REGION Network 93: 51.093 | n0093-ug7-el001-k30001_SN51 [3]
   RUNG wire#powerrail
      "FDBK_Error_n0093-ug7-el001-k30001_SN51_3"(Commissioning_bypass := "00_Commissioning"."n0093-ug7-el001-k30001_SN51", "FDBACK ERROR 1" := "FDBACK_=SG06+UG7.EL001-Q32801/Q32802".ERROR, "FDBACK ERROR 2" := "FDBACK_=SG06+UG7.EL001-Q32803/Q32804".ERROR, "FDBACK ERROR 3" := "FDBACK_=SG06+UG7.EL001-Q32901/Q32902".ERROR, "FDBACK ERROR 4" := "FDBACK_=SG06+UG7.EL001-Q32903/Q32904".ERROR, "FDBACK ERROR 5" :=, "FDBACK ERROR 6" :=, "FDBACK ERROR 7" :=, "FDBACK ERROR 8" :=, "Cumulative FDBACK" =>, "ERROR 1" => "03_FDBACK"."SG06+UG7.EL001-Q32802", "ERROR 2" => "03_FDBACK"."SG06+UG7.EL001-Q32804", "ERROR 3" => "03_FDBACK"."SG06+UG7.EL001-Q32902", "ERROR 4" => "03_FDBACK"."SG06+UG7.EL001-Q32904", "ERROR 5" =>, "ERROR 6" =>, "ERROR 7" =>, "ERROR 8" =>)
   END_RUNG
   // the same network as SCL:
   "FDBK_Error_n0093-ug7-el001-k30001_SN51_3"(Commissioning_bypass := "00_Commissioning"."n0093-ug7-el001-k30001_SN51",   // "03_FDBACK error"
                           "FDBACK ERROR 1" := "FDBACK_=SG06+UG7.EL001-Q32801/Q32802".ERROR,
                           "FDBACK ERROR 2" := "FDBACK_=SG06+UG7.EL001-Q32803/Q32804".ERROR,
                           "FDBACK ERROR 3" := "FDBACK_=SG06+UG7.EL001-Q32901/Q32902".ERROR,
                           "FDBACK ERROR 4" := "FDBACK_=SG06+UG7.EL001-Q32903/Q32904".ERROR,
                           "ERROR 1" => "03_FDBACK"."SG06+UG7.EL001-Q32802",
                           "ERROR 2" => "03_FDBACK"."SG06+UG7.EL001-Q32804",
                           "ERROR 3" => "03_FDBACK"."SG06+UG7.EL001-Q32902",
                           "ERROR 4" => "03_FDBACK"."SG06+UG7.EL001-Q32904");
END_REGION
END_FUNCTION

FUNCTION "07_Speed Control" : Void   // FC8, F_LAD
{ S7_Optimized_Access := 'TRUE' }
VERSION : 0.1
BEGIN

REGION Network 1: One network per sorter
END_REGION

REGION Network 2
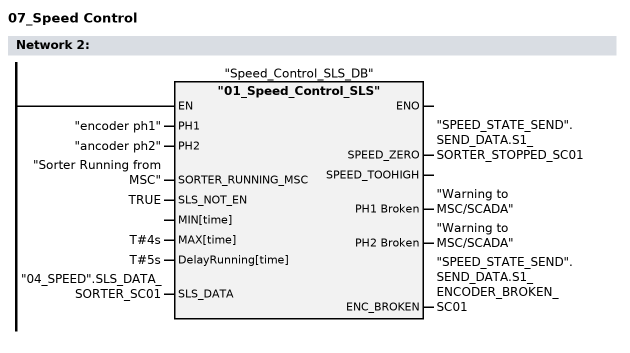
   RUNG wire#powerrail
      "Speed_Control_SLS_DB"(PH1 := "encoder ph1", PH2 := "ancoder ph2", SORTER_RUNNING_MSC := "Sorter Running from MSC", SLS_NOT_EN := TRUE, "MIN[time]" :=, "MAX[time]" := T#4s, "DelayRunning[time]" := T#5s, SLS_DATA := "04_SPEED".SLS_DATA_SORTER_SC01, SPEED_ZERO => "SPEED_STATE_SEND".SEND_DATA.S1_SORTER_STOPPED_SC01, SPEED_TOOHIGH =>, "PH1 Broken" => "Warning to MSC/SCADA", "PH2 Broken" => "Warning to MSC/SCADA", ENC_BROKEN => "SPEED_STATE_SEND".SEND_DATA.S1_ENCODER_BROKEN_SC01)
   END_RUNG
   // the same network as SCL:
   "Speed_Control_SLS_DB"(PH1 := "encoder ph1",   // "01_Speed_Control_SLS"
                          PH2 := "ancoder ph2",
                          SORTER_RUNNING_MSC := "Sorter Running from MSC",
                          SLS_NOT_EN := TRUE,
                          "MAX[time]" := T#4s,
                          "DelayRunning[time]" := T#5s,
                          SLS_DATA := "04_SPEED".SLS_DATA_SORTER_SC01,
                          SPEED_ZERO => "SPEED_STATE_SEND".SEND_DATA.S1_SORTER_STOPPED_SC01,
                          "PH1 Broken" => "Warning to MSC/SCADA",
                          "PH2 Broken" => "Warning to MSC/SCADA",
                          ENC_BROKEN => "SPEED_STATE_SEND".SEND_DATA.S1_ENCODER_BROKEN_SC01);
END_REGION
END_FUNCTION

FUNCTION "08_Gate Manager" : Void   // FC9, F_LAD
{ S7_Optimized_Access := 'TRUE' }
VERSION : 0.1
   VAR_TEMP
      temp_EXAMPLE_OPEN : Bool;
   END_VAR
BEGIN

REGION Network 1: Transfer Data from Speed Control
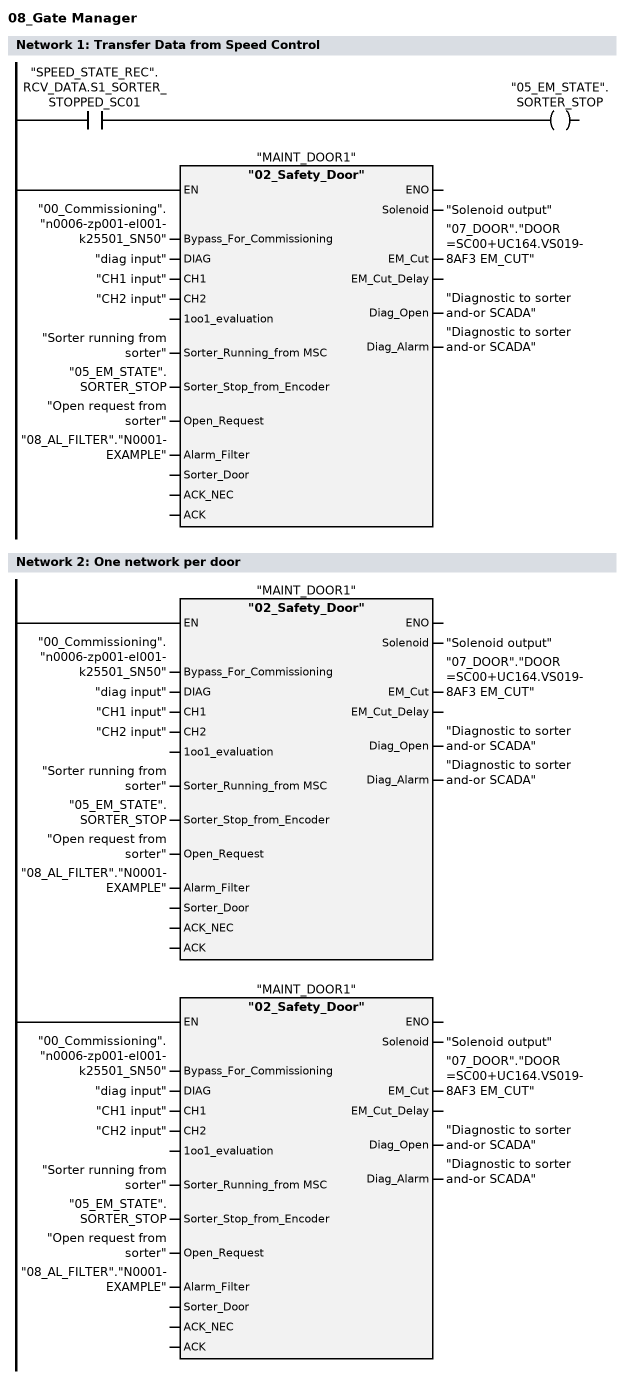
   RUNG wire#powerrail
      Contact( "SPEED_STATE_REC".RCV_DATA.S1_SORTER_STOPPED_SC01 )
      Coil( "05_EM_STATE".SORTER_STOP )
   END_RUNG
   RUNG wire#powerrail
      "MAINT_DOOR1"(Bypass_For_Commissioning := "00_Commissioning"."n0006-zp001-el001-k25501_SN50", DIAG := "diag input", CH1 := "CH1 input", CH2 := "CH2 input", "1oo1_evaluation" :=, "Sorter_Running_from MSC" := "Sorter running from sorter", Sorter_Stop_from_Encoder := "05_EM_STATE".SORTER_STOP, Open_Request := "Open request from sorter", Alarm_Filter := "08_AL_FILTER"."N0001-EXAMPLE", Sorter_Door :=, ACK_NEC :=, ACK :=, Solenoid => "Solenoid output", EM_Cut => "07_DOOR"."DOOR =SC00+UC164.VS019-8AF3 EM_CUT", EM_Cut_Delay =>, Diag_Open => "Diagnostic to sorter and-or SCADA", Diag_Alarm => "Diagnostic to sorter and-or SCADA")
   END_RUNG
   RUNG wire#powerrail
   END_RUNG
   // the same network as SCL:
   "05_EM_STATE".SORTER_STOP := "SPEED_STATE_REC".RCV_DATA.S1_SORTER_STOPPED_SC01;
   "MAINT_DOOR1"(Bypass_For_Commissioning := "00_Commissioning"."n0006-zp001-el001-k25501_SN50",   // "02_Safety_Door"
                 DIAG := "diag input",
                 CH1 := "CH1 input",
                 CH2 := "CH2 input",
                 "Sorter_Running_from MSC" := "Sorter running from sorter",
                 Sorter_Stop_from_Encoder := "05_EM_STATE".SORTER_STOP,
                 Open_Request := "Open request from sorter",
                 Alarm_Filter := "08_AL_FILTER"."N0001-EXAMPLE",
                 Solenoid => "Solenoid output",
                 EM_Cut => "07_DOOR"."DOOR =SC00+UC164.VS019-8AF3 EM_CUT",
                 Diag_Open => "Diagnostic to sorter and-or SCADA",
                 Diag_Alarm => "Diagnostic to sorter and-or SCADA");
END_REGION

REGION Network 2: One network per door
   RUNG wire#powerrail
      "MAINT_DOOR1"(Bypass_For_Commissioning := "00_Commissioning"."n0006-zp001-el001-k25501_SN50", DIAG := "diag input", CH1 := "CH1 input", CH2 := "CH2 input", "1oo1_evaluation" :=, "Sorter_Running_from MSC" := "Sorter running from sorter", Sorter_Stop_from_Encoder := "05_EM_STATE".SORTER_STOP, Open_Request := "Open request from sorter", Alarm_Filter := "08_AL_FILTER"."N0001-EXAMPLE", Sorter_Door :=, ACK_NEC :=, ACK :=, Solenoid => "Solenoid output", EM_Cut => "07_DOOR"."DOOR =SC00+UC164.VS019-8AF3 EM_CUT", EM_Cut_Delay =>, Diag_Open => "Diagnostic to sorter and-or SCADA", Diag_Alarm => "Diagnostic to sorter and-or SCADA")
   END_RUNG
   RUNG wire#powerrail
      "MAINT_DOOR1"(Bypass_For_Commissioning := "00_Commissioning"."n0006-zp001-el001-k25501_SN50", DIAG := "diag input", CH1 := "CH1 input", CH2 := "CH2 input", "1oo1_evaluation" :=, "Sorter_Running_from MSC" := "Sorter running from sorter", Sorter_Stop_from_Encoder := "05_EM_STATE".SORTER_STOP, Open_Request := "Open request from sorter", Alarm_Filter := "08_AL_FILTER"."N0001-EXAMPLE", Sorter_Door :=, ACK_NEC :=, ACK :=, Solenoid => "Solenoid output", EM_Cut => "07_DOOR"."DOOR =SC00+UC164.VS019-8AF3 EM_CUT", EM_Cut_Delay =>, Diag_Open => "Diagnostic to sorter and-or SCADA", Diag_Alarm => "Diagnostic to sorter and-or SCADA")
   END_RUNG
   // the same network as SCL:
   "MAINT_DOOR1"(Bypass_For_Commissioning := "00_Commissioning"."n0006-zp001-el001-k25501_SN50",   // "02_Safety_Door"
                 DIAG := "diag input",
                 CH1 := "CH1 input",
                 CH2 := "CH2 input",
                 "Sorter_Running_from MSC" := "Sorter running from sorter",
                 Sorter_Stop_from_Encoder := "05_EM_STATE".SORTER_STOP,
                 Open_Request := "Open request from sorter",
                 Alarm_Filter := "08_AL_FILTER"."N0001-EXAMPLE",
                 Solenoid => "Solenoid output",
                 EM_Cut => "07_DOOR"."DOOR =SC00+UC164.VS019-8AF3 EM_CUT",
                 Diag_Open => "Diagnostic to sorter and-or SCADA",
                 Diag_Alarm => "Diagnostic to sorter and-or SCADA");
   "MAINT_DOOR1"(Bypass_For_Commissioning := "00_Commissioning"."n0006-zp001-el001-k25501_SN50",   // "02_Safety_Door"
                 DIAG := "diag input",
                 CH1 := "CH1 input",
                 CH2 := "CH2 input",
                 "Sorter_Running_from MSC" := "Sorter running from sorter",
                 Sorter_Stop_from_Encoder := "05_EM_STATE".SORTER_STOP,
                 Open_Request := "Open request from sorter",
                 Alarm_Filter := "08_AL_FILTER"."N0001-EXAMPLE",
                 Solenoid => "Solenoid output",
                 EM_Cut => "07_DOOR"."DOOR =SC00+UC164.VS019-8AF3 EM_CUT",
                 Diag_Open => "Diagnostic to sorter and-or SCADA",
                 Diag_Alarm => "Diagnostic to sorter and-or SCADA");
END_REGION
END_FUNCTION

FUNCTION "00_Diagnostic PB" : Void   // FC10, STL
{ S7_Optimized_Access := 'TRUE' }
VERSION : 0.1
BEGIN

REGION Network 1: Example for coupler
   // each Push button has to be diagnosed, the output Q10005.0 is an example
         A     "01_PushButton"."SE01+ZP001.EL001-S31001_PB";
         O     "08_AL_FILTER"."N0001-EXAMPLE";
         =     "Tag_6";
END_REGION

REGION Network 2: Example for OPB
   // for each push button, use the following structure, the outputQ10005.0 is an example
         AN    "01_PushButton"."SE01+ZP001.EL001-S31001_PB";
         AN    "08_AL_FILTER"."N0001-EXAMPLE";
         =     "Tag_6";
END_REGION
END_FUNCTION

FUNCTION "01_DIagnostic Status" : Void   // FC11, STL
{ S7_Optimized_Access := 'TRUE' }
VERSION : 0.1
// Diagnostic for 
// sorter and zone status
// safety breaker status
BEGIN

REGION Network 1: Heartbeat
   // heartbeat sent to the Sorter Q0.0 is an example, normally the heartbeat is the first bit sent
         A     "Clock_0.5Hz";
         =     "Tag_3";
END_REGION

REGION Network 2: Sorter example
   // for each sorter, the ESTOP
   //SAFETYPLCEMERGENCYRE
         A     "ESTOP1_SORTER_CONV".Q;
         =     "Tag_1";

   //SAFETYPLCPOWERCUT
         A     "05_EM_STATE".POWER_CUT_SORTER;
         =     "Tag_4";
END_REGION

REGION Network 3: zone example
   // q10002.2  is an example
         A     "ESTOP1_EXAMPLE".Q;
         =     "Tag_5";
END_REGION

NETWORK
TITLE = Safety breaker
// Same logic as an E-STOP Push Button
END_FUNCTION

FUNCTION "02_Diagnostic Profinet" : Void   // FC12, LAD
{ S7_Optimized_Access := 'TRUE' }
VERSION : 0.1
   VAR_TEMP
      deviceState : Int;
      deviceState_1 : Int;
      deviceState_2 : Int;
      deviceState_3 : Int;
   END_VAR
BEGIN

REGION Network 1: MADA123 / One network per Subnet
   // LADDR:
   // You select the PROFINET IO or DP master system at the LADDR parameter by means of the hardware identifier.
   // 
   // The hardware identifier is available:
   // -Either in the Network view of the properties of the PROFINET IO or DP master system
   // -Or in the PLC tag table in the listed system constants with the data type HW_IOSYSTEM.
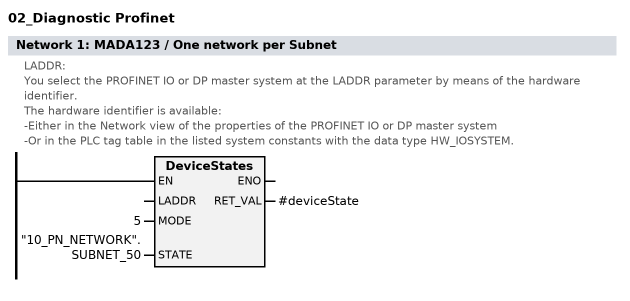
   // no SCL statement known for DeviceStates: written as a call
   #deviceState := DeviceStates(MODE := 5, STATE := "10_PN_NETWORK".SUBNET_50);
END_REGION
END_FUNCTION

FUNCTION "03_Diagnostic Nodes" : Void   // FC13, STL
{ S7_Optimized_Access := 'TRUE' }
VERSION : 0.1
BEGIN

REGION Network 1: One network per subnet
   // "00_Diagnostic_Profinet_DB"."Local~PROFINET_EXAMPLE"[x]
   // x = node number
   // 
   // Q10005.0 is an example
         AN    "10_PN_NETWORK".SUBNET_50[1];
         =     "Tag_6";
         A     "10_PN_NETWORK".SUBNET_50[1];
         =     "08_AL_FILTER"."N0001-EXAMPLE";
END_REGION
END_FUNCTION

FUNCTION "04_Diagnostic general alarms" : Void   // FC14, STL
{ S7_Optimized_Access := 'TRUE' }
VERSION : 0.1
// for other alarms diagnosed by the PLC
BEGIN
END_FUNCTION

FUNCTION "05_Diagnostic Feedback Error" : Void   // FC16, STL
{ S7_Optimized_Access := 'TRUE' }
VERSION : 0.1
BEGIN

REGION Network 1: Example
   // Each Feedbak error will be diagnosed in the same way as the Pushbuttons Q10005.0 is an example
         A     "03_FDBACK"."SC00+UC164.VS019-9QA4";
         =     "Tag_6";
END_REGION
END_FUNCTION

ORGANIZATION_BLOCK "Main"   // OB1, LAD, ProgramCycle
TITLE = "Main Program Sweep (Cycle)"
{ S7_Optimized_Access := 'TRUE' }
VERSION : 0.1
   VAR_INPUT
      Initial_Call : Bool;   // Initial call of this OB
      Remanence : Bool;   // =True, if remanent data are available
   END_VAR
BEGIN

REGION Network 1
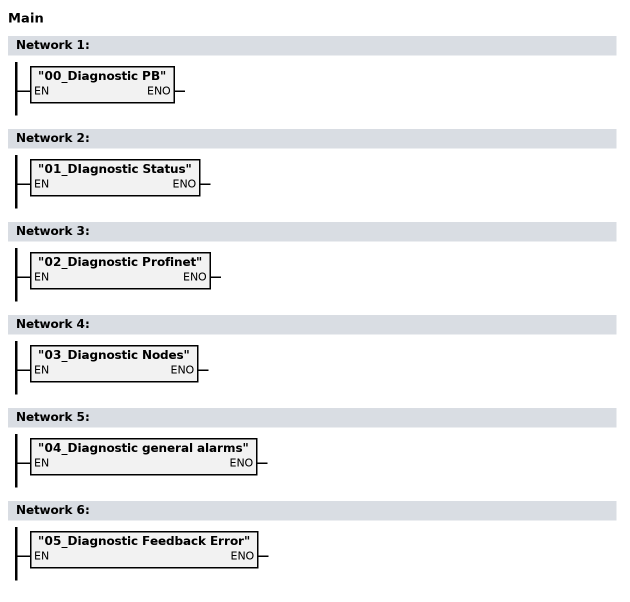
   RUNG wire#powerrail
      "00_Diagnostic PB"()
   END_RUNG
   // the same network as SCL:
   "00_Diagnostic PB"();
END_REGION

REGION Network 2
   RUNG wire#powerrail
      "01_DIagnostic Status"()
   END_RUNG
   // the same network as SCL:
   "01_DIagnostic Status"();
END_REGION

REGION Network 3
   RUNG wire#powerrail
      "02_Diagnostic Profinet"()
   END_RUNG
   // the same network as SCL:
   "02_Diagnostic Profinet"();
END_REGION

REGION Network 4
   RUNG wire#powerrail
      "03_Diagnostic Nodes"()
   END_RUNG
   // the same network as SCL:
   "03_Diagnostic Nodes"();
END_REGION

REGION Network 5
   RUNG wire#powerrail
      "04_Diagnostic general alarms"()
   END_RUNG
   // the same network as SCL:
   "04_Diagnostic general alarms"();
END_REGION

REGION Network 6
   RUNG wire#powerrail
      "05_Diagnostic Feedback Error"()
   END_RUNG
   // the same network as SCL:
   "05_Diagnostic Feedback Error"();
END_REGION
END_ORGANIZATION_BLOCK

ORGANIZATION_BLOCK "Programming error"   // OB121, LAD, ProgrammingError
{ S7_Optimized_Access := 'TRUE' }
VERSION : 0.1
   VAR_INPUT
      BlockNr : UInt;   // Number of causing block
      Reaction : USInt;   // 0:ignore, 1:substitute, 2:skip
      Fault_ID : Byte;   // Fault identifier
      BlockType : USInt;   // 16#01:OB, 16#02:FC, 16#03:FB, 16#04:SFC, 16#05:SFB, 16#06:DB: Type of block causing the error
      Area : USInt;   // Area where the error occured
      DBNr : DB_ANY;   // DB number if Area = DB or DI
      Csg_OBNr : OB_Any;   // Number of OB causing the error
      Csg_Prio : USInt;   // Priority of OB causing the error
      Width : USInt;   // 0:bit, 1:byte, 2:word, 3:dword, 4:lword
   END_VAR
BEGIN
END_ORGANIZATION_BLOCK

ORGANIZATION_BLOCK "IO access error"   // OB122, LAD, IOAccessError
{ S7_Optimized_Access := 'TRUE' }
VERSION : 0.1
   VAR_INPUT
      BlockNr : UInt;   // Number of causing block
      Reaction : USInt;   // 0:ignore, 1:substitute, 2:skip
      Fault_ID : Byte;   // 16#42:reading, 16#43:writing
      BlockType : USInt;   // 16#01:OB, 16#02:FC, 16#03:FB, 16#04:SFC, 16#05:SFB, 16#06:DB: Type of block causing the error
      Area : USInt;   // 16#81:I, 16#82:Q: IO area where the IOaccess error occured
      DBNr : DB_ANY;   // Reserved for system
      Csg_OBNr : OB_Any;   // Number of OB causing the error
      Csg_Prio : USInt;   // Priority of OB causing the error
      Width : USInt;   // 0:bit, 1:byte, 2:word, 3:dword, 4:lword
   END_VAR
BEGIN
END_ORGANIZATION_BLOCK

// folder: RTG_POST

FUNCTION "RTG2_POST" : Void   // FC15, LAD
{ S7_Optimized_Access := 'TRUE' }
VERSION : 0.1
BEGIN

REGION Network 1: Send the data to RTG1
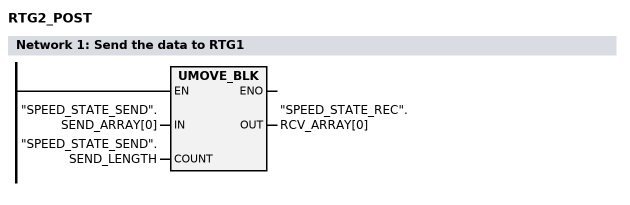
   UMOVE_BLK(IN := "SPEED_STATE_SEND".SEND_ARRAY[0],
             COUNT := "SPEED_STATE_SEND".SEND_LENGTH,
             OUT => "SPEED_STATE_REC".RCV_ARRAY[0]);
END_REGION
END_FUNCTION

FUNCTION "RTG1_POST" : Void   // FC17, LAD
{ S7_Optimized_Access := 'TRUE' }
VERSION : 0.1
BEGIN

REGION Network 1: Send the acknowledgment telegram to RTG2
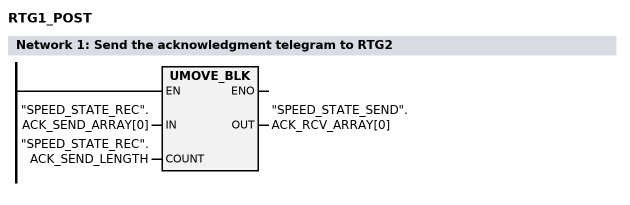
   UMOVE_BLK(IN := "SPEED_STATE_REC".ACK_SEND_ARRAY[0],
             COUNT := "SPEED_STATE_REC".ACK_SEND_LENGTH,
             OUT => "SPEED_STATE_SEND".ACK_RCV_ARRAY[0]);
END_REGION
END_FUNCTION